FUNCTION_BLOCK CbVtStatus (* This function is called in case of every page change - you can do e. g. initialisations ... *)
  (* Standard: ISO 11783-6; Description: This function is called in case of every page change - you can do e. g. initialisations ... *)
  (* Version 1.0, 2022-07-20, franz *)
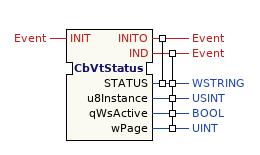
  EVENT_INPUT
    INIT; (* Service Initialization *)
  END_EVENT
  EVENT_OUTPUT
    INITO WITH STATUS; (* Initialization Confirm *)
    IND WITH STATUS, wPage, qWsActive, u8Instance; (* Indication from Resource *)
  END_EVENT
  VAR_OUTPUT
    STATUS : WSTRING; (* Service Status *)
    u8Instance : USINT; (* Identifier of the client instance *)
    qWsActive : BOOL; (* true, if the working set is active (displayed on screen) *)
    wPage : UINT; (* Contains the object ID of the open/last mask, or NULL object ID if unknown (ID_NULL = 0xFFFF) *)
  END_VAR
END_FUNCTION_BLOCK
